// TwinCAT 3 PLC project plc_kfe_gmd_vac
// ProgramVersion: 3.1.4022.3
// libraries:
//   L2SI Vacuum Library, * (SLAC)
//   LCLS General, * (SLAC)
//   PMPS, * (SLAC - LCLS)
//   Tc2_ControllerToolbox, * (Beckhoff Automation GmbH)
//   Tc2_MC2, * (Beckhoff Automation GmbH)
//   Tc2_Standard, * (Beckhoff Automation GmbH)
//   Tc2_System, * (Beckhoff Automation GmbH)
//   Tc2_Utilities, * (Beckhoff Automation GmbH)
//   Tc3_Module, * (Beckhoff Automation GmbH)
// project tree:
//   DUTs/ E_GasType.TcDUT (not stored), E_HomeState.TcDUT (not stored), E_MoveState.TcDUT (not stored), ST_HV.TcDUT (not stored), ST_PressureSensor.TcDUT (not stored), ST_VGP.TcDUT (not stored)
//   GVLs/ GVL_INJ.TcGVL (not stored), GVL_GMD.TcGVL (not stored), GVL_VARIABLES.TcGVL (not stored)
//   / PlcTask.TcTTO (not stored)
//   POUs/ FB_HighVoltage.TcPOU (not stored), FB_PressureTransducer.TcPOU (not stored), FB_RTD.TcPOU (not stored), FB_VGP.TcPOU (not stored), MAIN.TcPOU, PRG_DIAGNOSTIC.TcPOU (not stored), PRG_Gas_Selection.TcPOU (not stored), PRG_GMD.TcPOU (not stored), PRG_HV_ILK.TcPOU (not stored), PRG_INJ.TcPOU (not stored), PRG_PressureControl.TcPOU (not stored), PRG_Purge.TcPOU (not stored), PRG_VGP.TcPOU (not stored)
// real-time tasks:
//   TASK PlcTask: cycle T#10ms, priority 20, ADS port 350
//   TASK SimTask: cycle T#5ms, priority 21, ADS port 351
// motion (NC):
//   TASK NC-Task 1 SAF: cycle T#2ms, priority 4, ADS port 501
//   TASK NC-Task 1 SVB: cycle T#10ms, priority 8, ADS port 511
//   AXIS VGP_40 (id 3)
//     General: UnitName=steps
//     Velo: SlowManual=20, FastManual=30, Maximum=1800
//     OtherSettings: AllowMotionCmdToSlave=true
//     encoder EncType=4
//       EncPara: ScaleFactorNumerator=0.0390625, Inverse=true, MaxCount=#x0000ffff
//         SoftEndMinControl: Enable=true, Range=-20
//         SoftEndMaxControl: Enable=true, Range=1650
//         Inc: RefMode=2, RefSoftSyncMask=#x0000ffff
//     drive DrvType=24
//       Analog: VeloReferenz=2000, ScaleFactorActTorque=0.1
//       TimeComp: TaskDelayCycles=1
//     controller CtrType=1
//       CtrPara: PriorControlFactor=1
//         PosDiffControl: Range=50
//         Observer: BandWidth=20
// I/O:
//   DEVICE Device 1 (EtherCAT), AmsNetId 172.21.92.59.2.1
//     EK1200_00_00 [EK1200-5000 EtherCAT Power supply (2A E-Bus)]
//       EL3064_00_01 [EL3064 4Ch. Ana. Input 0-10V]
//       ES9070_00_02 [EL9070 Shield terminal]
//       EL1008_00_03 [EL1008 8Ch. Dig. Input 24V, 3ms]
//       ES9184_00_04 [EL9184 Potential Connection, 8 x 24V, 8 x Ground]
//       EL2008_00_05 [EL2008 8Ch. Dig. Output 24V, 0.5A]
//       EL2794_00_06 [EL2794 4Ch. Dig. Output 24V AC/DC, 2A, short-circuit-proof]
//       EL2202_00_07 [EL2202 2Ch. Dig. Output 24V, 0.5A]
//       EL6070_00_08 [EL6070 1Ch. Licensing-Terminal]
//       EL6695_00_09 [EL6695 EtherCAT Bridge terminal (Primary)]
//       EL6692_00_10 [EL6692 EtherCAT Bridge terminal (Primary)]
//       EK1110_00_11 [EK1110 EtherCAT extension]
//     EK1100_01_00 [EK1100 EtherCAT Coupler (2A E-Bus)]
//       EL2794_01_01 [EL2794 4Ch. Dig. Output 24V AC/DC, 2A, short-circuit-proof]
//       EL3068_01_02 [EL3068 8Ch. Ana. Input 0-10V]
//       EL3068_01_04 [EL3068 8Ch. Ana. Input 0-10V]
//       EL2794_01_05 [EL2794 4Ch. Dig. Output 24V AC/DC, 2A, short-circuit-proof]
//       EL2794_01_06 [EL2794 4Ch. Dig. Output 24V AC/DC, 2A, short-circuit-proof]
//       EL3068_01_07 [EL3068 8Ch. Ana. Input 0-10V]
//       EL3068_01_09 [EL3068 8Ch. Ana. Input 0-10V]
//       EL2794_01_10 [EL2794 4Ch. Dig. Output 24V AC/DC, 2A, short-circuit-proof]
//       EK1110_01_11 [EK1110 EtherCAT extension]
//     EK1100_02_00 [EK1100 EtherCAT Coupler (2A E-Bus)]
//       EL1004_02_01 [EL1004 4Ch. Dig. Input 24V, 3ms]
//       EL2004_02_02 [EL2004 4Ch. Dig. Output 24V, 0.5A]
//       EL1004_02_03 [EL1004 4Ch. Dig. Input 24V, 3ms]
//       EL1004_02_04 [EL1004 4Ch. Dig. Input 24V, 3ms]
//       EL2004_02_05 [EL2004 4Ch. Dig. Output 24V, 0.5A]
//       EL1004_02_06 [EL1004 4Ch. Dig. Input 24V, 3ms]
//       EL9410_02_07 [EL9410 E-Bus Power Supplier  (Diagnostics)]
//       EL1088_02_08 [EL1088 8Ch. Dig. Input 24V, 3ms, negative]
//       EL9187_02_09 [EL9187 Potential Connection, 8 x Ground]
//       EL2008_02_10 [EL2008 8Ch. Dig. Output 24V, 0.5A]
//       EL2088_02_10 [EL2088 8Ch. Dig. Output 24V, 0.5A, switching to negative] (disabled)
//       EL1088_02_11 [EL1088 8Ch. Dig. Input 24V, 3ms, negative]
//       EL1088_02_12 [EL1088 8Ch. Dig. Input 24V, 3ms, negative]
//       EL2088_02_14 [EL2088 8Ch. Dig. Output 24V, 0.5A, switching to negative] (disabled)
//       EL2008_02_14 [EL2008 8Ch. Dig. Output 24V, 0.5A]
//       EL1088_02_15 [EL1088 8Ch. Dig. Input 24V, 3ms, negative]
//       EL2004_02_16 [EL2004 4Ch. Dig. Output 24V, 0.5A]
//       EK1110_02_17 [EK1110 EtherCAT extension]
//     EK1100_03_00 [EK1100 EtherCAT Coupler (2A E-Bus)]
//       EL2794_03_01 [EL2794 4Ch. Dig. Output 24V AC/DC, 2A, short-circuit-proof]
//       EL3068_03_02 [EL3068 8Ch. Ana. Input 0-10V]
//       EL3068_03_04 [EL3068 8Ch. Ana. Input 0-10V]
//       EL2794_03_05 [EL2794 4Ch. Dig. Output 24V AC/DC, 2A, short-circuit-proof]
//       EL2794_03_06 [EL2794 4Ch. Dig. Output 24V AC/DC, 2A, short-circuit-proof]
//       EL1004_03_07 [EL1004 4Ch. Dig. Input 24V, 3ms]
//       EL9410_03_08 [EL9410 E-Bus Power Supplier  (Diagnostics)]
//       EL2212_03_09 [EL2212 2Ch. dig. output with overexcitation (24V DC, 2.5A, 10A Peak)]
//       Term 39 (EL9011) [EL9011 End Terminal]
//     EK1100_04_00 [EK1100 EtherCAT Coupler (2A E-Bus)]
//       ES2004_04_01 [EL2004 4Ch. Dig. Output 24V, 0.5A]
//       ES2004_04_02 [EL2004 4Ch. Dig. Output 24V, 0.5A]
//       ES3064_04_03 [EL3064 4Ch. Ana. Input 0-10V]
//       ES9070_04_04 [EL9070 Shield terminal]
//       ES3202_04_05 [EL3202 2Ch. Ana. Input PT100 (RTD)]
//       EL3054_04_06 [EL3054 4Ch. Ana. Input 4-20mA]
//       ES3064_04_07 [EL3064 4Ch. Ana. Input 0-10V]
//       ES9070_04_08 [EL9070 Shield terminal]
//       ES1008_04_09 [EL1008 8Ch. Dig. Input 24V, 3ms]
//       EL9184_04_10 [EL9184 Potential Connection, 8 x 24V, 8 x Ground]
//       ES2008_04_11 [EL2008 8Ch. Dig. Output 24V, 0.5A]
//       EL2794_04_12 [EL2794 4Ch. Dig. Output 24V AC/DC, 2A, short-circuit-proof]
//       EK1110_04_13 [EK1110 EtherCAT extension]
//     EP4374-0002_05_00 [EP4374-0002 2Ch. Ana. Input +/-10V, 0-10V, 0/4-20mA configurable; 2Ch. Ana. Output +/-10V, 0-10V, 0/4-20mA configurable]
//     EP5101-0011_05_01 [EP5101-0011 1Ch. Inc. Encoder 5V, D-SUB15]
//     EP7041-0002_05_02 [EP7041-0002 1Ch. Stepper motor output stage (50V, 5A)]
// variable links:
//   NC-Task 1 SAF/Axes/VGP_40 <-> Device 1 (EtherCAT)/EP5101-0011_05_01
//     Enc/Inputs/In/nDataIn1[0] <-> ENC Status compact/Counter value
//     Enc/Inputs/In/nDataIn2[0] <-> ENC Status compact/Latch value
//     Enc/Inputs/In/nState1 @bit 4 <-> ENC Status compact/Status/Counter overflow
//     Enc/Inputs/In/nState1 @bit 3 <-> ENC Status compact/Status/Counter underflow
//     Enc/Inputs/In/nState1 @bit 7 <-> ENC Status compact/Status/Extrapolation stall
//     Enc/Inputs/In/nState1 <-> ENC Status compact/Status/Latch C valid
//     Enc/Inputs/In/nState1 @bit 1 <-> ENC Status compact/Status/Latch extern valid
//     Enc/Inputs/In/nState1 @bit 6 <-> ENC Status compact/Status/Open circuit
//     Enc/Inputs/In/nState1 @bit 2 <-> ENC Status compact/Status/Set counter done
//     Enc/Inputs/In/nState1 @bit 5 <-> ENC Status compact/Status/Status of input status
//     Enc/Inputs/In/nState2 @bit 4 <-> ENC Status compact/Status/Status of extern latch
//     Enc/Inputs/In/nState2 <-> ENC Status compact/Status/Status of input A
//     Enc/Inputs/In/nState2 @bit 1 <-> ENC Status compact/Status/Status of input B
//     Enc/Inputs/In/nState2 @bit 2 <-> ENC Status compact/Status/Status of input C
//     Enc/Inputs/In/nState2 @bit 3 <-> ENC Status compact/Status/Status of input gate
//     Enc/Inputs/In/nState4 @bit 1 <-> WcState/InputToggle
//     Enc/Inputs/In/nState4 <-> WcState/WcState
//     Enc/Outputs/Out/nCtrl1 <-> ENC Control compact/Control/Enable latch C
//     Enc/Outputs/Out/nCtrl1 @bit 3 <-> ENC Control compact/Control/Enable latch extern on negative edge
//     Enc/Outputs/Out/nCtrl1 @bit 1 <-> ENC Control compact/Control/Enable latch extern on positive edge
//     Enc/Outputs/Out/nCtrl1 @bit 2 <-> ENC Control compact/Control/Set counter
//     Enc/Outputs/Out/nDataOut1[0] <-> ENC Control compact/Set counter value
//   NC-Task 1 SAF/Axes/VGP_40 <-> Device 1 (EtherCAT)/EP7041-0002_05_02
//     Drive/Inputs/In/nState1 @bit 3 <-> STM Status/Status/Error
//     Drive/Inputs/In/nState1 @bit 5 <-> STM Status/Status/Moving negative
//     Drive/Inputs/In/nState1 @bit 4 <-> STM Status/Status/Moving positive
//     Drive/Inputs/In/nState1 @bit 1 <-> STM Status/Status/Ready
//     Drive/Inputs/In/nState1 <-> STM Status/Status/Ready to enable
//     Drive/Inputs/In/nState1 @bit 6 <-> STM Status/Status/Torque reduced
//     Drive/Inputs/In/nState1 @bit 2 <-> STM Status/Status/Warning
//     Drive/Inputs/In/nState2 @bit 3 <-> STM Status/Status/Digital input 1
//     Drive/Inputs/In/nState2 @bit 4 <-> STM Status/Status/Digital input 2
//     Drive/Inputs/In/nState2 @bit 5 <-> STM Status/Status/Sync error
//     Drive/Inputs/In/nState2 @bit 7 <-> STM Status/Status/TxPDO Toggle
//     Drive/Inputs/In/nState4 @bit 1 <-> WcState/InputToggle
//     Drive/Inputs/In/nState4 <-> WcState/WcState
//     Drive/Outputs/Out/nCtrl1 <-> STM Control/Control/Enable
//     Drive/Outputs/Out/nCtrl1 @bit 2 <-> STM Control/Control/Reduce torque
//     Drive/Outputs/Out/nCtrl1 @bit 1 <-> STM Control/Control/Reset
//     Drive/Outputs/Out/nCtrl2 @bit 3 <-> STM Control/Control/Digital output 1
//     Drive/Outputs/Out/nDataOut2[0] <-> STM Velocity/Velocity
//   plc_kfe_gmd_vac/plc_kfe_gmd_vac Instance <-> Device 1 (EtherCAT)/EK1100_01_00/EL2794_01_01
//     PlcTask Outputs/GVL_GMD.fb_EM1K0_GMD_GCC_10.q_xHV_DIS <-> Channel 1/Output
//     PlcTask Outputs/GVL_GMD.fb_EM1K0_GMD_GCC_20.q_xHV_DIS <-> Channel 2/Output
//     PlcTask Outputs/GVL_GMD.fb_EM1K0_GMD_GCC_30.q_xHV_DIS <-> Channel 3/Output
//   plc_kfe_gmd_vac/plc_kfe_gmd_vac Instance <-> Device 1 (EtherCAT)/EK1100_01_00/EL2794_01_06
//     PlcTask Outputs/GVL_GMD.fb_EM1K0_GMD_GCC_50.q_xHV_DIS <-> Channel 1/Output
//     PlcTask Outputs/GVL_GMD.fb_EM1K0_GMD_GCC_60.q_xHV_DIS <-> Channel 2/Output
//   plc_kfe_gmd_vac/plc_kfe_gmd_vac Instance <-> Device 1 (EtherCAT)/EK1100_01_00/EL2794_01_10
//     PlcTask Outputs/GVL_GMD.fb_EM1K0_GMD_GCC_70.q_xHV_DIS <-> Channel 1/Output
//   plc_kfe_gmd_vac/plc_kfe_gmd_vac Instance <-> Device 1 (EtherCAT)/EK1100_01_00/EL3068_01_02
//     PlcTask Inputs/GVL_GMD.fb_EM1K0_GMD_GCC_10.i_iPRESS_R <-> AI Standard Channel 1/Value
//     PlcTask Inputs/GVL_GMD.fb_EM1K0_GMD_GCC_20.i_iPRESS_R <-> AI Standard Channel 2/Value
//     PlcTask Inputs/GVL_GMD.fb_EM1K0_GMD_GCC_30.i_iPRESS_R <-> AI Standard Channel 3/Value
//   plc_kfe_gmd_vac/plc_kfe_gmd_vac Instance <-> Device 1 (EtherCAT)/EK1100_01_00/EL3068_01_07
//     PlcTask Inputs/GVL_GMD.fb_EM1K0_GMD_GCC_50.i_iPRESS_R <-> AI Standard Channel 1/Value
//     PlcTask Inputs/GVL_GMD.fb_EM1K0_GMD_GCC_60.i_iPRESS_R <-> AI Standard Channel 3/Value
//     PlcTask Inputs/GVL_GMD.fb_EM1K0_GMD_GPI_70.i_iPRESS_R <-> AI Standard Channel 6/Value
//   plc_kfe_gmd_vac/plc_kfe_gmd_vac Instance <-> Device 1 (EtherCAT)/EK1100_01_00/EL3068_01_09
//     PlcTask Inputs/GVL_GMD.fb_EM1K0_GMD_GCC_70.i_iPRESS_R <-> AI Standard Channel 1/Value
//   plc_kfe_gmd_vac/plc_kfe_gmd_vac Instance <-> Device 1 (EtherCAT)/EK1100_02_00/EL1004_02_01
//     PlcTask Inputs/GVL_GMD.fb_EM1K0_GMD_VRC_10.i_xClsLS <-> Channel 2/Input
//     PlcTask Inputs/GVL_GMD.fb_EM1K0_GMD_VRC_20.i_xClsLS <-> Channel 4/Input
//     PlcTask Inputs/GVL_GMD.fb_EM1K0_GMD_VRC_10.i_xOpnLS <-> Channel 1/Input
//     PlcTask Inputs/GVL_GMD.fb_EM1K0_GMD_VRC_20.i_xOpnLS <-> Channel 3/Input
//   plc_kfe_gmd_vac/plc_kfe_gmd_vac Instance <-> Device 1 (EtherCAT)/EK1100_02_00/EL1004_02_03
//     PlcTask Inputs/GVL_GMD.fb_EM1K0_GMD_VRC_30.i_xClsLS <-> Channel 2/Input
//     PlcTask Inputs/GVL_GMD.fb_EM1K0_GMD_VRC_30.i_xOpnLS <-> Channel 1/Input
//   plc_kfe_gmd_vac/plc_kfe_gmd_vac Instance <-> Device 1 (EtherCAT)/EK1100_02_00/EL1004_02_04
//     PlcTask Inputs/GVL_GMD.fb_EM1K0_GMD_VRC_50.i_xClsLS <-> Channel 2/Input
//     PlcTask Inputs/GVL_GMD.fb_EM1K0_GMD_VRC_60.i_xClsLS <-> Channel 4/Input
//     PlcTask Inputs/GVL_GMD.fb_EM1K0_GMD_VRC_50.i_xOpnLS <-> Channel 1/Input
//     PlcTask Inputs/GVL_GMD.fb_EM1K0_GMD_VRC_60.i_xOpnLS <-> Channel 3/Input
//   plc_kfe_gmd_vac/plc_kfe_gmd_vac Instance <-> Device 1 (EtherCAT)/EK1100_02_00/EL1004_02_06
//     PlcTask Inputs/GVL_GMD.fb_EM1K0_GMD_VRC_70.i_xClsLS <-> Channel 2/Input
//     PlcTask Inputs/GVL_GMD.fb_EM1K0_GMD_VRC_70.i_xOpnLS <-> Channel 1/Input
//   plc_kfe_gmd_vac/plc_kfe_gmd_vac Instance <-> Device 1 (EtherCAT)/EK1100_02_00/EL1088_02_08
//     PlcTask Inputs/GVL_GMD.fb_EM1K0_GMD_PTM_10.i_xAtSpd <-> Channel 1/Input
//     PlcTask Inputs/GVL_GMD.fb_EM1K0_GMD_PTM_20.i_xAtSpd <-> Channel 3/Input
//   plc_kfe_gmd_vac/plc_kfe_gmd_vac Instance <-> Device 1 (EtherCAT)/EK1100_02_00/EL1088_02_11
//     PlcTask Inputs/GVL_GMD.fb_EM1K0_GMD_PTM_30.i_xAtSpd <-> Channel 1/Input
//     PlcTask Inputs/GVL_GMD.fb_EM1K0_GMD_PTM_40.i_xAtSpd <-> Channel 3/Input
//   plc_kfe_gmd_vac/plc_kfe_gmd_vac Instance <-> Device 1 (EtherCAT)/EK1100_02_00/EL1088_02_12
//     PlcTask Inputs/GVL_GMD.fb_EM1K0_GMD_PTM_50.i_xAtSpd <-> Channel 1/Input
//     PlcTask Inputs/GVL_GMD.fb_EM1K0_GMD_PTM_60.i_xAtSpd <-> Channel 3/Input
//   plc_kfe_gmd_vac/plc_kfe_gmd_vac Instance <-> Device 1 (EtherCAT)/EK1100_02_00/EL1088_02_15
//     PlcTask Inputs/GVL_GMD.fb_EM1K0_GMD_PTM_70.i_xAtSpd <-> Channel 1/Input
//   plc_kfe_gmd_vac/plc_kfe_gmd_vac Instance <-> Device 1 (EtherCAT)/EK1100_02_00/EL2004_02_02
//     PlcTask Outputs/GVL_GMD.fb_EM1K0_GMD_VRC_10.q_xOPN_DO <-> Channel 1/Output
//     PlcTask Outputs/GVL_GMD.fb_EM1K0_GMD_VRC_20.q_xOPN_DO <-> Channel 3/Output
//     PlcTask Outputs/GVL_GMD.fb_EM1K0_GMD_VRC_30.q_xOPN_DO <-> Channel 2/Output
//     PlcTask Outputs/GVL_GMD.fb_EM1K0_GMD_VRC_30.q_xOPN_DO <-> Channel 4/Output
//   plc_kfe_gmd_vac/plc_kfe_gmd_vac Instance <-> Device 1 (EtherCAT)/EK1100_02_00/EL2004_02_05
//     PlcTask Outputs/GVL_GMD.fb_EM1K0_GMD_VRC_50.q_xOPN_DO <-> Channel 1/Output
//     PlcTask Outputs/GVL_GMD.fb_EM1K0_GMD_VRC_60.q_xOPN_DO <-> Channel 3/Output
//     PlcTask Outputs/GVL_GMD.fb_EM1K0_GMD_VRC_70.q_xOPN_DO <-> Channel 2/Output
//     PlcTask Outputs/GVL_GMD.fb_EM1K0_GMD_VRC_70.q_xOPN_DO <-> Channel 4/Output
//   plc_kfe_gmd_vac/plc_kfe_gmd_vac Instance <-> Device 1 (EtherCAT)/EK1100_02_00/EL2004_02_16
//     PlcTask Outputs/GVL_GMD.fb_EM1K0_GMD_VRC_10.q_xOPN_DO <-> Channel 1/Output
//     PlcTask Outputs/GVL_GMD.fb_EM1K0_GMD_VRC_20.q_xOPN_DO <-> Channel 3/Output
//     PlcTask Outputs/GVL_GMD.fb_EM1K0_GMD_VRC_50.q_xOPN_DO <-> Channel 2/Output
//     PlcTask Outputs/GVL_GMD.fb_EM1K0_GMD_VRC_60.q_xOPN_DO <-> Channel 4/Output
//   plc_kfe_gmd_vac/plc_kfe_gmd_vac Instance <-> Device 1 (EtherCAT)/EK1100_02_00/EL2008_02_10
//     PlcTask Outputs/GVL_GMD.fb_EM1K0_GMD_PTM_{10..40 step 10}.q_RunDO <-> Channel {1..4}/Output  (4 links)
//   plc_kfe_gmd_vac/plc_kfe_gmd_vac Instance <-> Device 1 (EtherCAT)/EK1100_02_00/EL2008_02_14
//     PlcTask Outputs/GVL_GMD.fb_EM1K0_GMD_PTM_50.q_RunDO <-> Channel 1/Output
//     PlcTask Outputs/GVL_GMD.fb_EM1K0_GMD_PTM_60.q_RunDO <-> Channel 2/Output
//     PlcTask Outputs/GVL_GMD.fb_EM1K0_GMD_PTM_70.q_RunDO <-> Channel 3/Output
//   plc_kfe_gmd_vac/plc_kfe_gmd_vac Instance <-> Device 1 (EtherCAT)/EK1100_02_00/EL2088_02_10
//     PlcTask Outputs/GVL_GMD.fb_EM1K0_GMD_PTM_{10..40 step 10}.q_RunDO <-> Channel {1..4}/Output  (4 links)
//   plc_kfe_gmd_vac/plc_kfe_gmd_vac Instance <-> Device 1 (EtherCAT)/EK1100_02_00/EL2088_02_14
//     PlcTask Outputs/GVL_GMD.fb_EM1K0_GMD_PTM_50.q_RunDO <-> Channel 1/Output
//     PlcTask Outputs/GVL_GMD.fb_EM1K0_GMD_PTM_60.q_RunDO <-> Channel 2/Output
//     PlcTask Outputs/GVL_GMD.fb_EM1K0_GMD_PTM_70.q_RunDO <-> Channel 3/Output
//   plc_kfe_gmd_vac/plc_kfe_gmd_vac Instance <-> Device 1 (EtherCAT)/EK1100_03_00/EL1004_03_07
//     PlcTask Inputs/GVL_GMD.fb_EM1K0_GMD_PRT_40.i_xAlarmOK <-> Channel 2/Input
//     PlcTask Inputs/GVL_GMD.fb_EM1K0_GMD_PRT_40.i_xIsRun <-> Channel 1/Input
//   plc_kfe_gmd_vac/plc_kfe_gmd_vac Instance <-> Device 1 (EtherCAT)/EK1100_03_00/EL2794_03_01
//     PlcTask Outputs/GVL_GMD.fb_EM1K0_GMD_GCC_40.q_xHV_DIS <-> Channel 2/Output
//   plc_kfe_gmd_vac/plc_kfe_gmd_vac Instance <-> Device 1 (EtherCAT)/EK1100_03_00/EL2794_03_06
//     PlcTask Outputs/GVL_GMD.fb_EM1K0_GMD_PRT_40.q_xRemote <-> Channel 2/Output
//     PlcTask Outputs/GVL_GMD.fb_EM1K0_GMD_PRT_40.q_xRunDo <-> Channel 1/Output
//   plc_kfe_gmd_vac/plc_kfe_gmd_vac Instance <-> Device 1 (EtherCAT)/EK1100_03_00/EL3068_03_02
//     PlcTask Inputs/GVL_GMD.fb_EM1K0_GMD_GCC_40.i_iPRESS_R <-> AI Standard Channel 3/Value
//     PlcTask Inputs/GVL_GMD.fb_EM1K0_GMD_GPI_10.i_iPRESS_R <-> AI Standard Channel 6/Value
//     PlcTask Inputs/GVL_GMD.fb_EM1K0_GMD_GPI_40.i_iPRESS_R <-> AI Standard Channel 5/Value
//   plc_kfe_gmd_vac/plc_kfe_gmd_vac Instance <-> Device 1 (EtherCAT)/EK1100_04_00/EL3054_04_06
//     PlcTask Inputs/GVL_INJ.GFM_{83..86}.i_iPRESS_R <-> AI Standard Channel {1..4}/Value  (4 links)
//   plc_kfe_gmd_vac/plc_kfe_gmd_vac Instance <-> Device 1 (EtherCAT)/EK1100_04_00/ES2004_04_01
//     PlcTask Outputs/GVL_INJ.VVC_80.q_xOPN_DO <-> Channel 1/Output
//     PlcTask Outputs/GVL_INJ.VVC_81.q_xOPN_DO <-> Channel 3/Output
//     PlcTask Outputs/GVL_INJ.VVC_82.q_xOPN_DO <-> Channel 4/Output
//   plc_kfe_gmd_vac/plc_kfe_gmd_vac Instance <-> Device 1 (EtherCAT)/EK1100_04_00/ES2004_04_02
//     PlcTask Outputs/GVL_INJ.VVC_{83..86}.q_xOPN_DO <-> Channel {1..4}/Output  (4 links)
//   plc_kfe_gmd_vac/plc_kfe_gmd_vac Instance <-> Device 1 (EtherCAT)/EK1100_04_00/ES3202_04_05
//     PlcTask Inputs/GVL_INJ.RTD.bError <-> RTD Inputs Channel 1/Status/Error
//     PlcTask Inputs/GVL_INJ.RTD.bOverrange <-> RTD Inputs Channel 1/Status/Overrange
//     PlcTask Inputs/GVL_INJ.RTD.bUnderrange <-> RTD Inputs Channel 1/Status/Underrange
//     PlcTask Inputs/GVL_INJ.RTD.iRaw <-> RTD Inputs Channel 1/Value
//   plc_kfe_gmd_vac/plc_kfe_gmd_vac Instance <-> Device 1 (EtherCAT)/EK1200_00_00/EL1008_00_03
//     PlcTask Inputs/GVL_GMD.fb_EM1K0_GMD_PTM_{10..70 step 10}.i_xFault <-> Channel {1..7}/Input  (7 links)
//   plc_kfe_gmd_vac/plc_kfe_gmd_vac Instance <-> Device 1 (EtherCAT)/EK1200_00_00/EL2008_00_05
//     PlcTask Outputs/GVL_GMD.fb_EM1K0_GMD_PTM_{10..70 step 10}.q_RunDO <-> Channel {1..7}/Output  (7 links)
//   plc_kfe_gmd_vac/plc_kfe_gmd_vac Instance <-> Device 1 (EtherCAT)/EP4374-0002_05_00
//     PlcTask Inputs/GVL_INJ.GCM_80.i_iPRESS_R <-> AI Inputs Channel 1/Value
//     PlcTask Outputs/GVL_INJ.VCN_40.q_iRawPosition <-> AO Outputs Channel 3/Analog output

// ---- POUs/MAIN.TcPOU
PROGRAM MAIN
VAR
	
END_VAR

PRG_DIAGNOSTIC();
PRG_GMD();


(*INJ*)
PRG_INJ();
PRG_PressureControl();
//PRG_Purge();
//call orther PRG

// instaniate the RTD and HV

END_PROGRAM
